TYPE Fraction :
STRUCT
	Numerator : LREAL;
	Denominator : LREAL;
END_STRUCT
END_TYPE

(* stored: Version 1.1.0.1
   DUT Fraction: Id {9fe5d316-993a-0d8a-0313-85b3ff3b56bb} *)
